// TIA Portal V17 export
// export: Created 2022-10-14T12:26:27.5573765Z, ExportSetting WithDefaults, DisplayName Totally Integrated Automation Portal, DisplayVersion V17 Update 4, DisplayName TIA Portal Openness, DisplayVersion V17 Update 4, DisplayName TIA Portal Version Control Interface, DisplayVersion V17, DisplayName SINAMICS Startdrive Advanced, DisplayVersion V17 Update2, DisplayName SINAMICS Startdrive G130, G150, S120, S150, SINAMICS MV, S210, DisplayVersion V17 Update2, DisplayName SINAMICS Startdrive G110M, G120, G120C, G120D, G120P, G115D, DisplayVersion V17 Update2, DisplayName STEP 7 Professional, DisplayVersion V17 Update 4, DisplayName STEP 7 Safety, DisplayVersion V17, DisplayName WinCC Advanced / Unified PC, DisplayVersion V17 Update 4
FUNCTION "Inkr_per_Pulse" : Void   // FC500, FBD
{ S7_Optimized_Access := 'TRUE' }
VERSION : 0.1
// M.alsouki
// stored: AutoNumber false, IsIECCheckEnabled false, SetENOAutomatically false, UDAEnableTagReadback false
   VAR_INPUT
      Reset : Bool;
      Pulse : Bool;
      Up : Bool;
      down : Bool;
      Inkr_Up : Real;
      Inkr_Down : Real;
      Limit_Up : Real;
      Limit_Down : Real;
   END_VAR
   VAR_IN_OUT
      Value : Real;
   END_VAR
BEGIN

REGION Network 1: Nullen
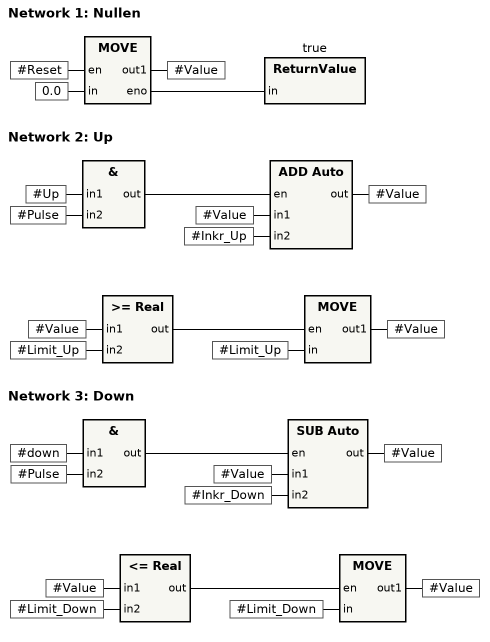
   IF #Reset THEN
       #Value := 0.0;
       ENO := true;
       RETURN;
   END_IF;
END_REGION

REGION Network 2: Up
   IF #Up AND #Pulse THEN #Value := #Value + #Inkr_Up; END_IF;
   IF #Value >= #Limit_Up THEN #Value := #Limit_Up; END_IF;
END_REGION

REGION Network 3: Down
   IF #down AND #Pulse THEN #Value := #Value - #Inkr_Down; END_IF;
   IF #Value <= #Limit_Down THEN #Value := #Limit_Down; END_IF;
END_REGION
END_FUNCTION
